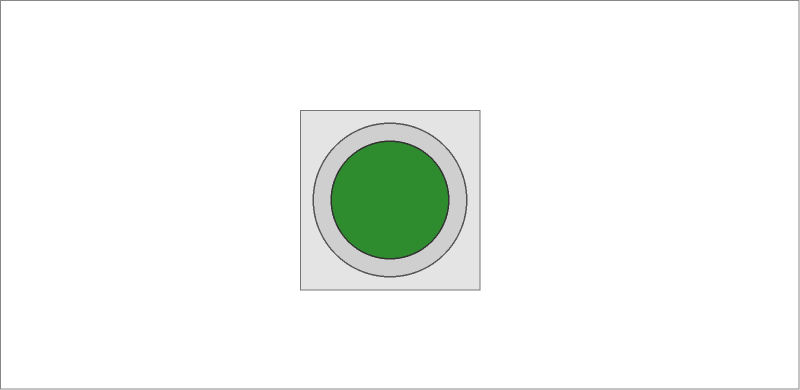
VISUALIZATION VisuDigitalOutControl  // 800x390
VAR_IN_OUT
	fbManualControler	: FB_ManualController ;
END_VAR
    PushSwitch (300,110 180x180), variable: fbManualControler.pDevDigitalOut^.bCmdOn, behaviour: TOGGLE, style: Switch-PushSwitch-Green
END_VISUALIZATION

(* stored: Version 1.1.0.1, ProductVersion 3.1.4024.11
   Visu VisuDigitalOutControl: Id {b4d6e9db-b1e9-0669-04c2-7a8e94b601ad} *)
